// TIA Portal V18 export
DATA_BLOCK "Tests_Executing"   // DB97
{ S7_Optimized_Access := 'TRUE' }
VERSION : 0.1
// stored: AutoNumber true, DBAccessibleFromOPCUA true, IsOnlyStoredInLoadMemory false, IsRetainMemResEnabled false, IsWriteProtectedInAS false, MemoryReserve 100
   VAR
      Test01_Enable : Bool;   // Z2 Relative Motion Test Enable
      Test01_Start : Bool;   // Z2 Relative Motion Test Start
      Test01_End : Bool;   // Z2 Relative Motion Test End
   END_VAR
BEGIN
END_DATA_BLOCK
